(* IEC 61131-3 sources: eCockpitGit/test_project/src/%F%02 System/%F%03 LoadSaveManager/%POU%FB_LoadSave/%F%Load/%F%Structure, 7 files *)

(* ---- %METH%compareKeyName.st ---- *)
//Returns true if the inputted string is the same as the read string
METHOD compareKeyName : EStructType
VAR_INPUT
	name				:POINTER TO EASCII;
END_VAR

(*%!%__DELIMITER__%!%*)
compareKeyName		:=		reader.compareKeyName(name:=name);

(* ---- %METH%exportSelection.st ---- *)
//This method outputs the start address and size of the currently selected object
//True when ok
// |**Version**|**Author**| **Date** |**Changes**
// | 1         | NSN      | 04-06-18 | Creation
METHOD exportSelection : BOOL
VAR_OUTPUT
	position		:POINTER TO EASCII;
	size			:DWORD;
END_VAR
(*%!%__DELIMITER__%!%*)
exportSelection		:=		reader.exportSelection(position=>position,size=>size);

(* ---- %METH%exportValue.st ---- *)
//This method outputs the start address and size of the currently selected value
//True when ok
// |**Version**|**Author**| **Date** |**Changes**
// | 1         | NSN      | 04-06-18 | Creation
METHOD exportValue : BOOL
VAR_OUTPUT
	position		:POINTER TO EASCII;
	size			:DWORD;
END_VAR
(*%!%__DELIMITER__%!%*)
exportValue		:=		reader.exportValue(position=>position,size=>size);

(* ---- %METH%findKey.st ---- *)
//This method finds the key of the given name in the object
//Returns cursor to where it was before if no tag is found
// |**Version**|**Author**| **Date** |**Changes**
// | 1         | NSN      | 04-06-18 | Creation
METHOD findKey : EStructType
VAR_INPUT
	name			:POINTER TO EASCII;		//Address of the name to find, only input string address or zero terminated byte array
END_VAR
(*%!%__DELIMITER__%!%*)
findKey		:=		reader.findKey(name:=name);

(* ---- %METH%readKeyName.st ---- *)
METHOD readKeyName : BOOL
VAR_INPUT
	name			:POINTER TO EASCII;		//Address of the name to find, only input string address or zero terminated byte array
	lenMax			:DWORD;
END_VAR
VAR_OUTPUT
	len				:WORD;
END_VAR
(*%!%__DELIMITER__%!%*)
readKeyName		:=		reader.readKeyName(name:=name,lenMax:=lenMax,len=>len);

(* ---- %METH%readKeyNameChar.st ---- *)
//This method returns the character of a given position from the key name
//Returns null if out of range
//1 is the first character, 0 is also the first character
METHOD readKeyNameChar : EASCII
VAR_INPUT
	charNum			:WORD;		//Character number
END_VAR
(*%!%__DELIMITER__%!%*)
readKeyNameChar		:=		reader.readKeyNameChar(charNum:=charNum);

(* ---- %METH%readKeyNameLevel.st ---- *)
METHOD readKeyNameLevel : BOOL
VAR_INPUT
	name			:POINTER TO EASCII;		//Address of the name to find, only input string address or zero terminated byte array
	lenMax			:DWORD;					//Max lenght of string value
	level			:BYTE;					//The level to get from
END_VAR
VAR_OUTPUT
	len				:WORD;					//Actual lenght of string value
END_VAR
(*%!%__DELIMITER__%!%*)
readKeyNameLevel		:=		reader.readKeyNameLevel(name:=name,lenMax:=lenMax,level:=level,len=>len);
